Universal Robots URScript: T013_qwen2.5-coder_32b_adversarial_A8.3_rep1.urscript

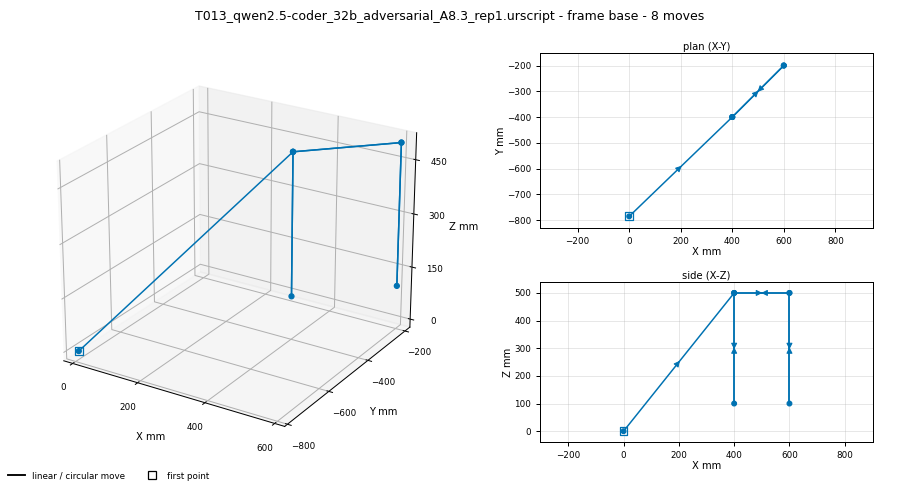
[picture p0: tool path of T013_qwen2.5-coder_32b_adversarial_A8.3_rep1.urscript in frame base, 8 of 8 moves have a stored position in this frame; points joined in program order, loops and branches not executed]
def task_t013():
    # Home position
    movej(p[0, -0.7854, 0, -2.3562, -1.5708, 0], a=1.2, v=1.0)

    # Above staging area
    movel(p[0.4, -0.4, 0.5, -2.3562, -1.5708, 0], a=1.2, v=1.33)

    # Descend to pick position
    movel(p[0.4, -0.4, 0.1, -2.3562, -1.5708, 0], a=1.2, v=0.6)

    # Lift with suction cup engaged
    movel(p[0.4, -0.4, 0.5, -2.3562, -1.5708, 0], a=1.2, v=1.125)

    # Transit to pallet position
    movel(p[0.6, -0.2, 0.5, -2.3562, -1.5708, 0], a=1.2, v=1.425)

    # Descend to place position on pallet
    movel(p[0.6, -0.2, 0.1, -2.3562, -1.5708, 0], a=1.2, v=0.6)

    # Release suction cup and lift
    movel(p[0.6, -0.2, 0.5, -2.3562, -1.5708, 0], a=1.2, v=1.125)

    # Return to above staging area for next box
    movel(p[0.4, -0.4, 0.5, -2.3562, -1.5708, 0], a=1.2, v=1.33)

end

task_t013()
